Staubli VAL3: remGetOneHere.pgx

program remGetOneHere(string& sArgs[] (dimensions=1), string& sReturn[] (dimensions=1))
  local joint jHere
  local num nPos
begin
  // Return just one position.
  //
  logMsg("call remGetOneHere")
  call remCalcHereSph()
  jHere=herej()
  sReturn="GETONEPOS "+sArgs+" "
  switch sArgs
    case "X"
      nPos=nXHere
    break
    case "Y"
      nPos=nYHere
    break
    case "Z"
      nPos=nZHere
    break
    case "RX"
      nPos=nRXHere
    break
    case "RY"
      nPos=nRYHere
    break
    case "RZ"
      nPos=nRZHere
    break
    case "AZI"
      nPos=nAzHere
    break
    case "ELE"
      nPos=nElHere
    break
    case "RAD"
      nPos=nRHere
    break
    case "J1"
      nPos=jHere.j1
    break
    case "J2"
      nPos=jHere.j2
    break
    case "J3"
      nPos=jHere.j3
    break
    case "J4"
      nPos=jHere.j4
    break
    case "J5"
      nPos=jHere.j5
    break
    case "J6"
      nPos=jHere.j6
    break
    default
      call remErrInvalid("GETONEPOS",sArgs,sReturn)
    break
  endSwitch
  sReturn=sReturn+toString(sNumConv,nPos)
end
